FUNCTION_BLOCK FB_OnlineChangeMovePadding
VAR
	aPadding: ARRAY[1..512] OF UDINT;
END_VAR

END_FUNCTION_BLOCK

(* stored: Version 1.1.0.1
   POU FB_OnlineChangeMovePadding: Id {b9be61c7-0f84-4204-86dd-d6a6604c25b6}, SpecialFunc None *)
